(* Logix 5000 project; controller Lavado_Tapado Emulate 5570 rev 32.11; software revision 32.00 *)

TASK MainTask (continuous, watchdog 500 ms) : MainProgram

MODULES
   Local : Emulate 5570 (ICP 2, rev 32.11)
END_MODULES

VAR_GLOBAL   (* controller tags *)
   ACT_LLT_AlineadorLlenado : BOOL;   // Orden NX de extensión del alineador.
   ACT_LLT_Banda : BOOL := 1;   // Orden NX de encendido de la banda.
   ACT_LLT_BoquillaLlenado : BOOL;   // Orden NX de descenso de la boquilla.
   ACT_LLT_BorrarBotella : BOOL;   // Orden NX de borrar el CAD sin tapa.
   ACT_LLT_DetencionLlenado : BOOL;   // Orden NX de retención de botellas.
   ACT_LLT_NuevaBotella : BOOL;   // Orden NX de crear el CAD con tapa.
   ACT_LLT_PosicionamientoTapado : DINT;   // Consigna numérica NX del carrusel en grados.
   ACT_LLT_Remachadora : BOOL;   // Orden NX de descenso de la remachadora.
   CMD_LLT_Inicio : BOOL := 1;   // Botón momentáneo de Inicio desde Studio 5000.
   CMD_LLT_Parada : BOOL;   // Botón momentáneo de Parada; abandona el automático.
   CMD_LLT_Reinicio : BOOL;   // Botón momentáneo de Reinicio con prioridad máxima.
   CNT_LLT_BotellasGrupo : DINT; {access None}   // Conteo numérico del grupo de botellas.
   ET_LLT_000_Inicial : BOOL; {access None}   // Etapa 0 inicial y reiniciada.
   ET_LLT_010_Automatico : BOOL := 1; {access None}   // Etapa 10 de automático concurrente.
   ET_LLT_090_Parada : BOOL; {access None}   // Etapa 90 de parada sin reanudación.
   ET_LLT_100_Admision : BOOL := 1; {access None}   // Etapa 100 de admisión y conteo.
   ET_LLT_110_Posicionamiento : BOOL; {access None}   // Etapa 110 de posicionamiento durante 2 s.
   ET_LLT_120_Alineacion : BOOL; {access None}   // Etapa 120 de extensión del alineador.
   ET_LLT_130_DescensoBoquilla : BOOL; {access None}   // Etapa 130 de descenso de boquilla.
   ET_LLT_140_Llenado : BOOL; {access None}   // Etapa 140 de llenado durante 2 s.
   ET_LLT_150_RetiradaBoquilla : BOOL; {access None}   // Etapa 150 de subida de boquilla.
   ET_LLT_160_RetiradaAlineacion : BOOL; {access None}   // Etapa 160 de retracción del alineador.
   ET_LLT_170_Transferencia : BOOL; {access None}   // Etapa 170 de transferencia del grupo.
   ET_LLT_200_EsperaPrimeraBotella : BOOL; {access None}   // Etapa 200 de espera de primera botella en carrusel.
   ET_LLT_210_PrimerIndexado : BOOL; {access None}   // Etapa 210 de primer indexado.
   ET_LLT_220_BorrarPrimera : BOOL; {access None}   // Etapa 220 de borrar primera botella.
   ET_LLT_222_CrearPrimera : BOOL; {access None}   // Etapa 222 de crear primera botella con tapa.
   ET_LLT_230_SegundoIndexado : BOOL; {access None}   // Etapa 230 de segundo indexado.
   ET_LLT_240_Borrar : BOOL; {access None}   // Etapa 240 de borrado en rama paralela.
   ET_LLT_241_Crear : BOOL; {access None}   // Etapa 241 de creación en rama paralela.
   ET_LLT_242_TapadoListo : BOOL; {access None}   // Etapa 242 de tapado listo.
   ET_LLT_250_BajarRemachadora : BOOL; {access None}   // Etapa 250 de descenso de remachadora.
   ET_LLT_251_SubirRemachadora : BOOL; {access None}   // Etapa 251 de subida de remachadora.
   ET_LLT_252_RemachadoListo : BOOL; {access None}   // Etapa 252 de remachado listo.
   ET_LLT_260_IndexadoSincronizado : BOOL := 1; {access None}   // Etapa 260 de indexado sincronizado.
   FL_LLT_ContadorEntrada : BOOL; {access None}   // Pulso de flanco ascendente del sensor de entrada.
   FL_LLT_CuartaBotella : BOOL; {access None}   // Pulso de cuarto evento aceptado.
   IDX_LLT_Carrusel : DINT; {access None}   // Índice cíclico del carrusel de 0 a 4.
   M_LLT_ConteoHabilitado : BOOL := 1; {access None}   // Ventana de conteo exclusiva de etapa 100.
   M_LLT_ReinicioCumplido : BOOL := 1; {access None}   // Memoria que exige Reinicio después de Parada antes de aceptar Inicio.
   M_LLT_RemacheVioAusencia : BOOL := 1; {access None}   // Memoria de ausencia previa del sensor de remache.
   M_LLT_TapadoVioAusencia : BOOL := 1; {access None}   // Memoria de ausencia previa del sensor de tapado.
   MEM_LLT_ContadorEntradaPrev : BOOL; {access None}   // Memoria ONS global del sensor de entrada; evita contar un nivel ya activo al entrar en admisión.
   PAR_LLT_BotellasGrupo : DINT := 4;   // Cantidad objetivo de botellas por grupo.
   PAR_LLT_PasoCarrusel_deg : DINT := -72;   // Paso angular lógico del carrusel.
   PAR_LLT_PosicionesCarrusel : DINT := 5;   // Cantidad de posiciones lógicas del carrusel.
   PAR_LLT_T_Llenado_ms : DINT := 2000;   // Preset de llenado en milisegundos.
   PAR_LLT_T_Posicionamiento_ms : DINT := 2000;   // Preset de posicionamiento en milisegundos.
   SE_LLT_AgregarTapa : BOOL;   // Botella presente en la estación de tapado.
   SE_LLT_AlineacionLlenadoExtendido : BOOL;   // Alineador completamente extendido.
   SE_LLT_AlineacionLlenadoRetraido : BOOL := 1;   // Alineador completamente retraído.
   SE_LLT_BoquillaAbajo : BOOL;   // Boquilla completamente abajo.
   SE_LLT_BoquillaArriba : BOOL := 1;   // Boquilla completamente arriba.
   SE_LLT_ContadorEntrada : BOOL;   // Botella frente al sensor de entrada; se cuenta solo por flanco en admisión.
   SE_LLT_DeteccionBotellaTapado : BOOL;   // Botella disponible en la entrada del carrusel.
   SE_LLT_ParadaRemache : BOOL := 1;   // Botella presente en la estación de remache.
   SE_LLT_RemachadoraAbajo : BOOL;   // Remachadora completamente abajo.
   SE_LLT_RemachadoraArriba : BOOL := 1;   // Remachadora completamente arriba.
   SE_LLT_SinDetencion : BOOL := 1;   // Tope retirado y paso libre; no existe sensor de tope extendido.
   SP_LLT_Carrusel_deg : DINT; {access None}   // Consigna interna vigente del carrusel en grados.
   TM_LLT_Llenado : TIMER := (PRE := 2000); {access None}   // Temporizador de llenado de 2 s.
   TM_LLT_Posicionamiento : TIMER := (PRE := 2000); {access None}   // Temporizador de posicionamiento de 2 s.
   TR_LLT_t00 : BOOL; {access None}   // Snapshot de la transición t00; se evalúa antes de actualizar etapas.
   TR_LLT_t10 : BOOL; {access None}   // Snapshot de la transición t10; se evalúa antes de actualizar etapas.
   TR_LLT_t100 : BOOL; {access None}   // Snapshot de la transición t100; se evalúa antes de actualizar etapas.
   TR_LLT_t110 : BOOL; {access None}   // Snapshot de la transición t110; se evalúa antes de actualizar etapas.
   TR_LLT_t120 : BOOL; {access None}   // Snapshot de la transición t120; se evalúa antes de actualizar etapas.
   TR_LLT_t130 : BOOL; {access None}   // Snapshot de la transición t130; se evalúa antes de actualizar etapas.
   TR_LLT_t140 : BOOL; {access None}   // Snapshot de la transición t140; se evalúa antes de actualizar etapas.
   TR_LLT_t150 : BOOL; {access None}   // Snapshot de la transición t150; se evalúa antes de actualizar etapas.
   TR_LLT_t160 : BOOL; {access None}   // Snapshot de la transición t160; se evalúa antes de actualizar etapas.
   TR_LLT_t170 : BOOL; {access None}   // Snapshot de la transición t170; se evalúa antes de actualizar etapas.
   TR_LLT_t200 : BOOL; {access None}   // Snapshot de la transición t200; se evalúa antes de actualizar etapas.
   TR_LLT_t210 : BOOL; {access None}   // Snapshot de la transición t210; se evalúa antes de actualizar etapas.
   TR_LLT_t220 : BOOL; {access None}   // Snapshot de la transición t220; se evalúa antes de actualizar etapas.
   TR_LLT_t220a : BOOL; {access None}   // Snapshot de la transición t220a; se evalúa antes de actualizar etapas.
   TR_LLT_t230 : BOOL; {access None}   // Snapshot de la transición t230; se evalúa antes de actualizar etapas.
   TR_LLT_t240 : BOOL; {access None}   // Snapshot de la transición t240; se evalúa antes de actualizar etapas.
   TR_LLT_t240a : BOOL; {access None}   // Snapshot de la transición t240a; se evalúa antes de actualizar etapas.
   TR_LLT_t250 : BOOL; {access None}   // Snapshot de la transición t250; se evalúa antes de actualizar etapas.
   TR_LLT_t250a : BOOL; {access None}   // Snapshot de la transición t250a; se evalúa antes de actualizar etapas.
   TR_LLT_t260 : BOOL; {access None}   // Snapshot de la transición t260; se evalúa antes de actualizar etapas.
   TR_LLT_t261 : BOOL; {access None}   // Snapshot de la transición t261; se evalúa antes de actualizar etapas.
   TR_LLT_t90 : BOOL; {access None}   // Snapshot de la transición t90; se evalúa antes de actualizar etapas.
END_VAR

PROGRAM MainProgram   (* main routine MainRoutine *)

ROUTINE MainRoutine   (* ladder *)
// Despacha seis rutinas simplificadas en orden determinista.
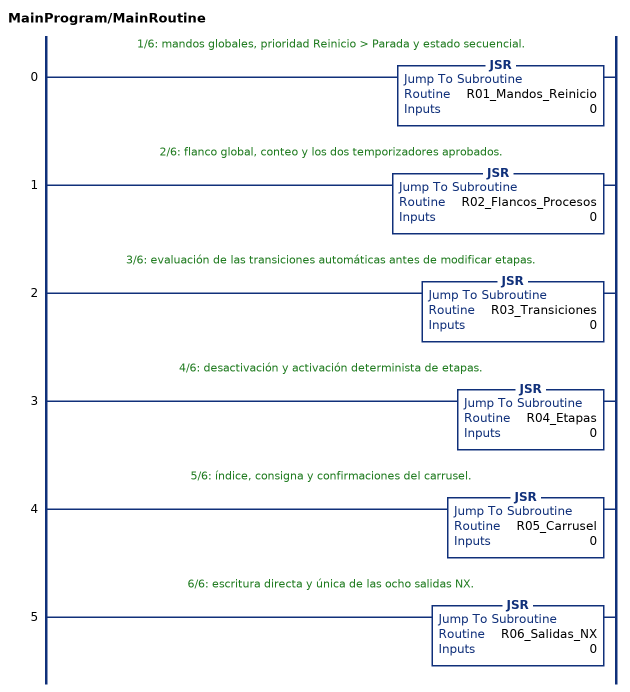
   // 1/6: mandos globales, prioridad Reinicio > Parada y estado secuencial.
   0: JSR(R01_Mandos_Reinicio,0);
   // 2/6: flanco global, conteo y los dos temporizadores aprobados.
   1: JSR(R02_Flancos_Procesos,0);
   // 3/6: evaluación de las transiciones automáticas antes de modificar etapas.
   2: JSR(R03_Transiciones,0);
   // 4/6: desactivación y activación determinista de etapas.
   3: JSR(R04_Etapas,0);
   // 5/6: índice, consigna y confirmaciones del carrusel.
   4: JSR(R05_Carrusel,0);
   // 6/6: escritura directa y única de las ocho salidas NX.
   5: JSR(R06_Salidas_NX,0);
END_ROUTINE

ROUTINE R01_Mandos_Reinicio   (* ladder *)
// Mandos globales y retorno simple al estado inicial sin escribir actuadores.
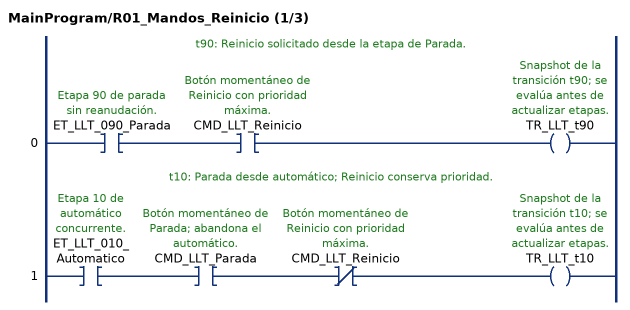
   // t90: Reinicio solicitado desde la etapa de Parada.
   0: XIC(ET_LLT_090_Parada)XIC(CMD_LLT_Reinicio)OTE(TR_LLT_t90);
   // t10: Parada desde automático; Reinicio conserva prioridad.
   1: XIC(ET_LLT_010_Automatico)XIC(CMD_LLT_Parada)XIO(CMD_LLT_Reinicio)OTE(TR_LLT_t10);
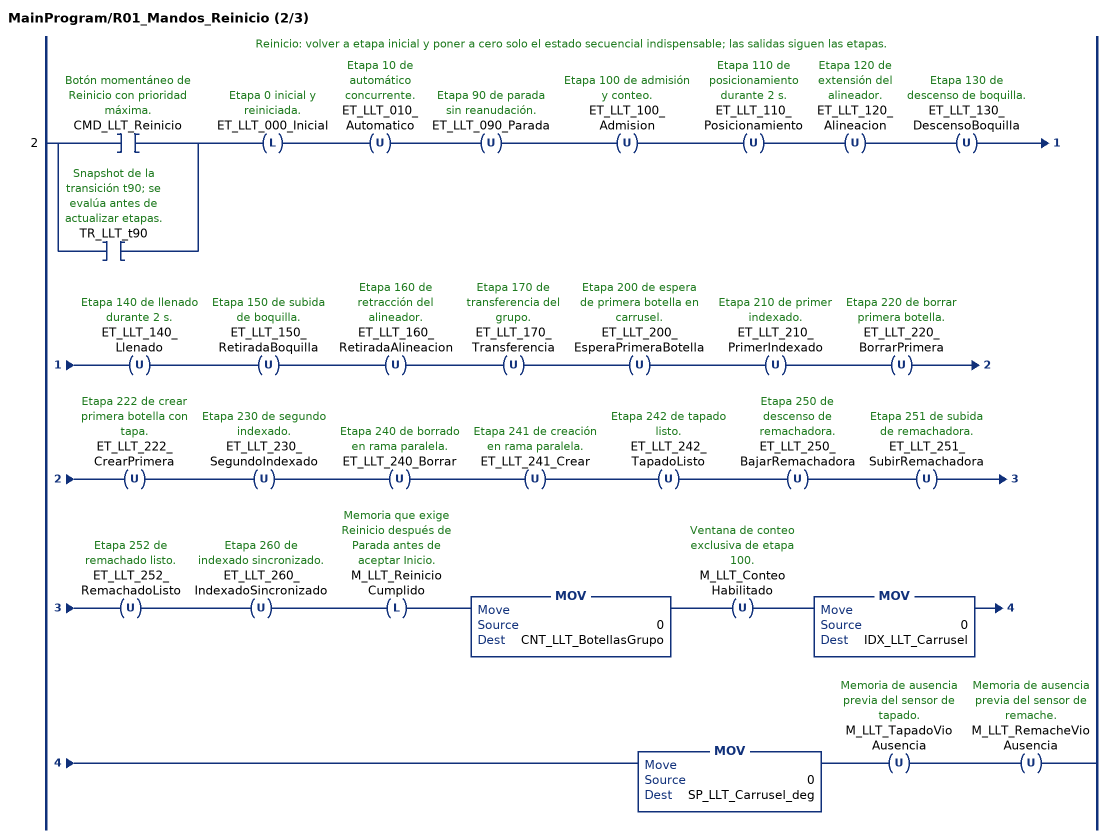
   // Reinicio: volver a etapa inicial y poner a cero solo el estado secuencial indispensable; las salidas siguen las etapas.
   2: [XIC(CMD_LLT_Reinicio) ,XIC(TR_LLT_t90) ]OTL(ET_LLT_000_Inicial)OTU(ET_LLT_010_Automatico)OTU(ET_LLT_090_Parada)OTU(ET_LLT_100_Admision)OTU(ET_LLT_110_Posicionamiento)OTU(ET_LLT_120_Alineacion)OTU(ET_LLT_130_DescensoBoquilla)OTU(ET_LLT_140_Llenado)OTU(ET_LLT_150_RetiradaBoquilla)OTU(ET_LLT_160_RetiradaAlineacion)OTU(ET_LLT_170_Transferencia)OTU(ET_LLT_200_EsperaPrimeraBotella)OTU(ET_LLT_210_PrimerIndexado)OTU(ET_LLT_220_BorrarPrimera)OTU(ET_LLT_222_CrearPrimera)OTU(ET_LLT_230_SegundoIndexado)OTU(ET_LLT_240_Borrar)OTU(ET_LLT_241_Crear)OTU(ET_LLT_242_TapadoListo)OTU(ET_LLT_250_BajarRemachadora)OTU(ET_LLT_251_SubirRemachadora)OTU(ET_LLT_252_RemachadoListo)OTU(ET_LLT_260_IndexadoSincronizado)OTL(M_LLT_ReinicioCumplido)MOV(0,CNT_LLT_BotellasGrupo)OTU(M_LLT_ConteoHabilitado)MOV(0,IDX_LLT_Carrusel)MOV(0,SP_LLT_Carrusel_deg)OTU(M_LLT_TapadoVioAusencia)OTU(M_LLT_RemacheVioAusencia);
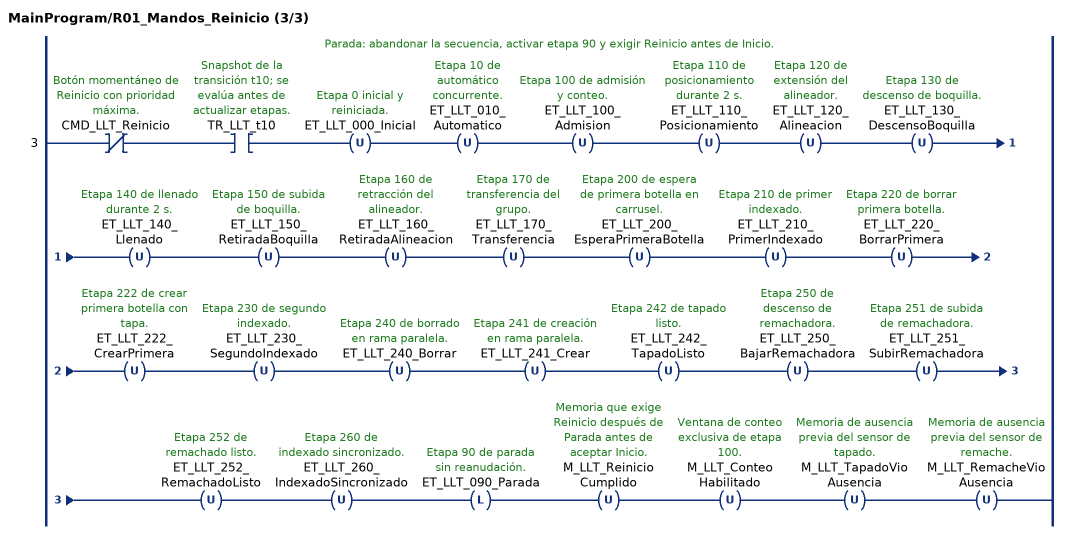
   // Parada: abandonar la secuencia, activar etapa 90 y exigir Reinicio antes de Inicio.
   3: XIO(CMD_LLT_Reinicio)XIC(TR_LLT_t10)OTU(ET_LLT_000_Inicial)OTU(ET_LLT_010_Automatico)OTU(ET_LLT_100_Admision)OTU(ET_LLT_110_Posicionamiento)OTU(ET_LLT_120_Alineacion)OTU(ET_LLT_130_DescensoBoquilla)OTU(ET_LLT_140_Llenado)OTU(ET_LLT_150_RetiradaBoquilla)OTU(ET_LLT_160_RetiradaAlineacion)OTU(ET_LLT_170_Transferencia)OTU(ET_LLT_200_EsperaPrimeraBotella)OTU(ET_LLT_210_PrimerIndexado)OTU(ET_LLT_220_BorrarPrimera)OTU(ET_LLT_222_CrearPrimera)OTU(ET_LLT_230_SegundoIndexado)OTU(ET_LLT_240_Borrar)OTU(ET_LLT_241_Crear)OTU(ET_LLT_242_TapadoListo)OTU(ET_LLT_250_BajarRemachadora)OTU(ET_LLT_251_SubirRemachadora)OTU(ET_LLT_252_RemachadoListo)OTU(ET_LLT_260_IndexadoSincronizado)OTL(ET_LLT_090_Parada)OTU(M_LLT_ReinicioCumplido)OTU(M_LLT_ConteoHabilitado)OTU(M_LLT_TapadoVioAusencia)OTU(M_LLT_RemacheVioAusencia);
END_ROUTINE

ROUTINE R02_Flancos_Procesos   (* ladder *)
// Flanco global, conteo de cuatro y únicamente dos TON.
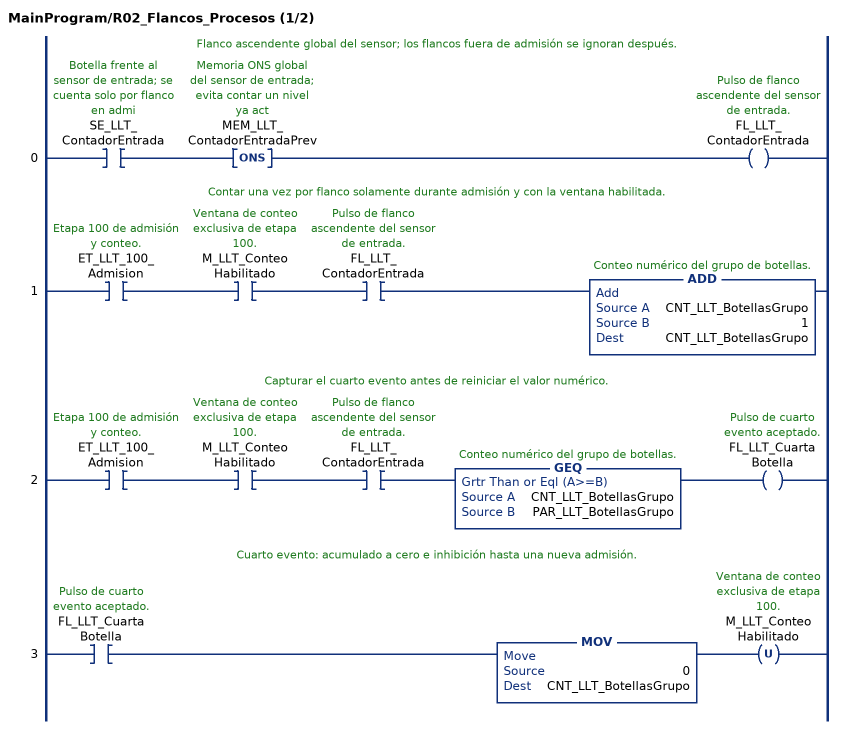
   // Flanco ascendente global del sensor; los flancos fuera de admisión se ignoran después.
   0: XIC(SE_LLT_ContadorEntrada)ONS(MEM_LLT_ContadorEntradaPrev)OTE(FL_LLT_ContadorEntrada);
   // Contar una vez por flanco solamente durante admisión y con la ventana habilitada.
   1: XIC(ET_LLT_100_Admision)XIC(M_LLT_ConteoHabilitado)XIC(FL_LLT_ContadorEntrada)ADD(CNT_LLT_BotellasGrupo,1,CNT_LLT_BotellasGrupo);
   // Capturar el cuarto evento antes de reiniciar el valor numérico.
   2: XIC(ET_LLT_100_Admision)XIC(M_LLT_ConteoHabilitado)XIC(FL_LLT_ContadorEntrada)GEQ(CNT_LLT_BotellasGrupo,PAR_LLT_BotellasGrupo)OTE(FL_LLT_CuartaBotella);
   // Cuarto evento: acumulado a cero e inhibición hasta una nueva admisión.
   3: XIC(FL_LLT_CuartaBotella)MOV(0,CNT_LLT_BotellasGrupo)OTU(M_LLT_ConteoHabilitado);
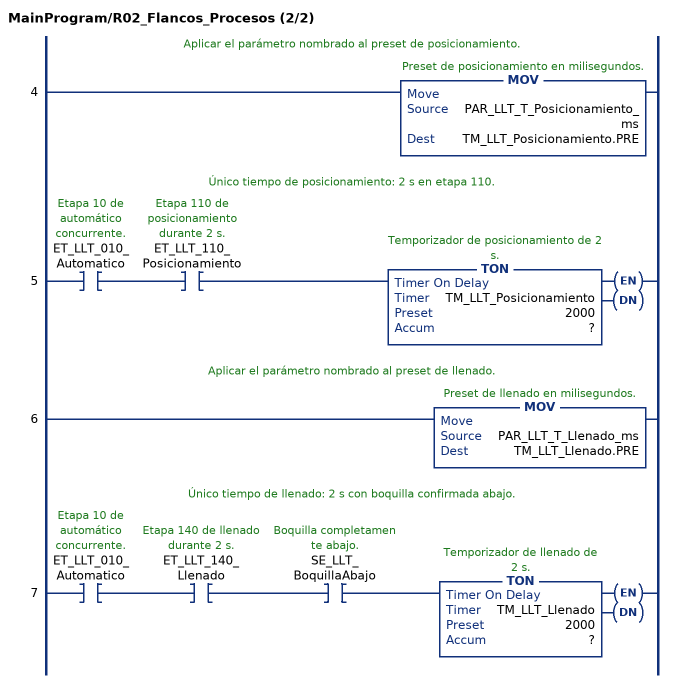
   // Aplicar el parámetro nombrado al preset de posicionamiento.
   4: MOV(PAR_LLT_T_Posicionamiento_ms,TM_LLT_Posicionamiento.PRE);
   // Único tiempo de posicionamiento: 2 s en etapa 110.
   5: XIC(ET_LLT_010_Automatico)XIC(ET_LLT_110_Posicionamiento)TON(TM_LLT_Posicionamiento,?,?);
   // Aplicar el parámetro nombrado al preset de llenado.
   6: MOV(PAR_LLT_T_Llenado_ms,TM_LLT_Llenado.PRE);
   // Único tiempo de llenado: 2 s con boquilla confirmada abajo.
   7: XIC(ET_LLT_010_Automatico)XIC(ET_LLT_140_Llenado)XIC(SE_LLT_BoquillaAbajo)TON(TM_LLT_Llenado,?,?);
END_ROUTINE

ROUTINE R03_Transiciones   (* ladder *)
// Evalúa las veinte transiciones automáticas; t10 y t90 se resuelven antes en mandos.
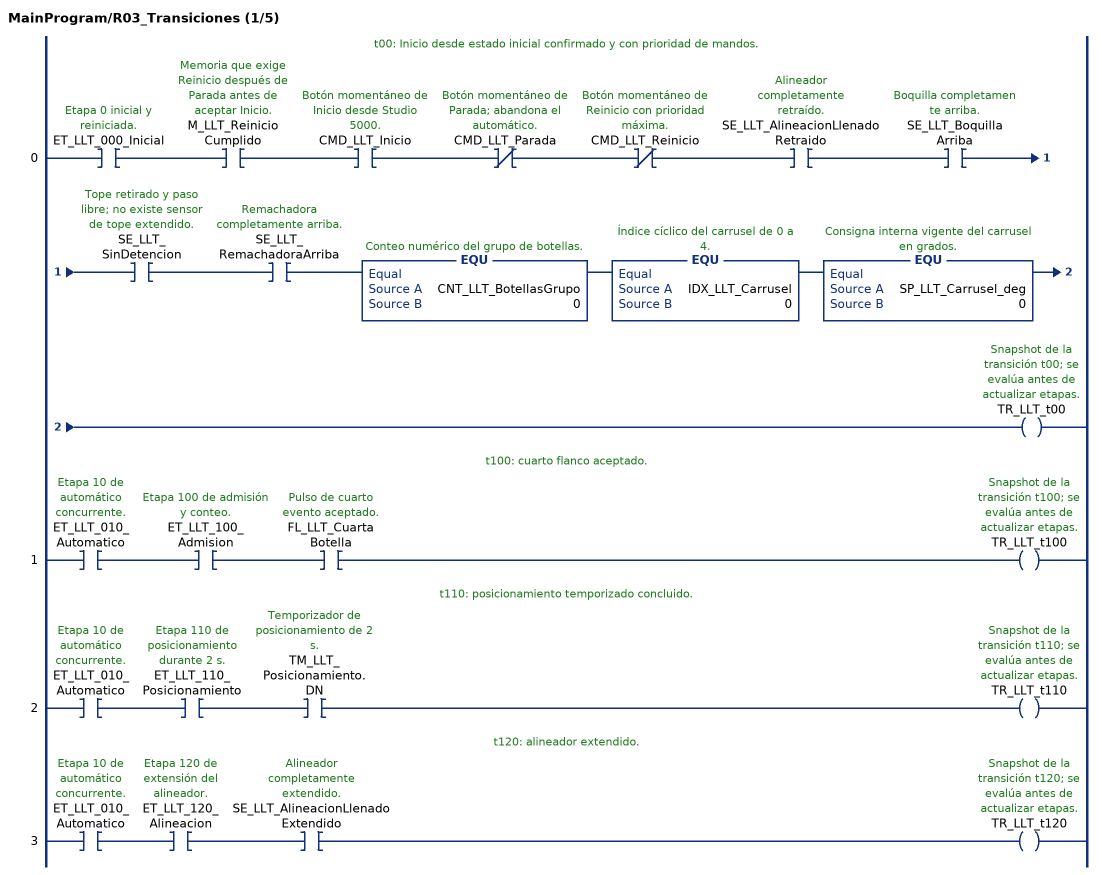
   // t00: Inicio desde estado inicial confirmado y con prioridad de mandos.
   0: XIC(ET_LLT_000_Inicial)XIC(M_LLT_ReinicioCumplido)XIC(CMD_LLT_Inicio)XIO(CMD_LLT_Parada)XIO(CMD_LLT_Reinicio)XIC(SE_LLT_AlineacionLlenadoRetraido)XIC(SE_LLT_BoquillaArriba)XIC(SE_LLT_SinDetencion)XIC(SE_LLT_RemachadoraArriba)EQU(CNT_LLT_BotellasGrupo,0)EQU(IDX_LLT_Carrusel,0)EQU(SP_LLT_Carrusel_deg,0)OTE(TR_LLT_t00);
   // t100: cuarto flanco aceptado.
   1: XIC(ET_LLT_010_Automatico)XIC(ET_LLT_100_Admision)XIC(FL_LLT_CuartaBotella)OTE(TR_LLT_t100);
   // t110: posicionamiento temporizado concluido.
   2: XIC(ET_LLT_010_Automatico)XIC(ET_LLT_110_Posicionamiento)XIC(TM_LLT_Posicionamiento.DN)OTE(TR_LLT_t110);
   // t120: alineador extendido.
   3: XIC(ET_LLT_010_Automatico)XIC(ET_LLT_120_Alineacion)XIC(SE_LLT_AlineacionLlenadoExtendido)OTE(TR_LLT_t120);
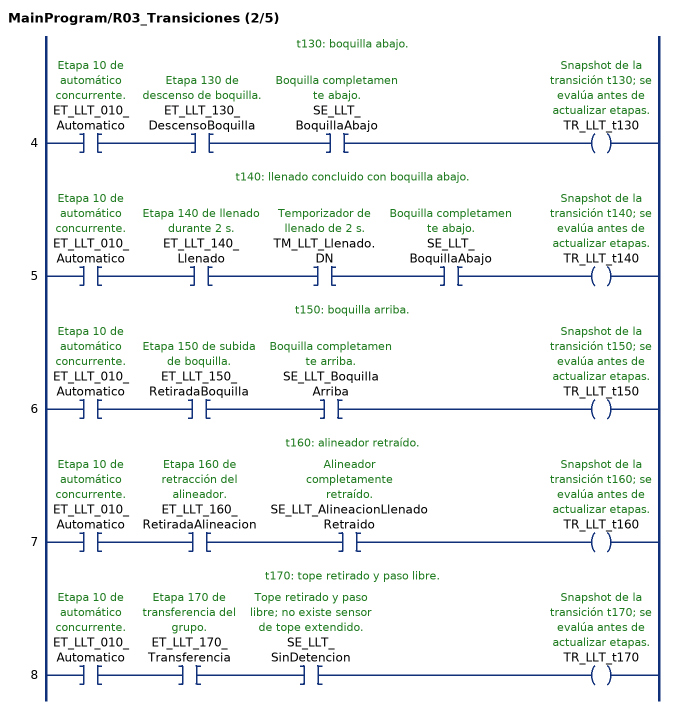
   // t130: boquilla abajo.
   4: XIC(ET_LLT_010_Automatico)XIC(ET_LLT_130_DescensoBoquilla)XIC(SE_LLT_BoquillaAbajo)OTE(TR_LLT_t130);
   // t140: llenado concluido con boquilla abajo.
   5: XIC(ET_LLT_010_Automatico)XIC(ET_LLT_140_Llenado)XIC(TM_LLT_Llenado.DN)XIC(SE_LLT_BoquillaAbajo)OTE(TR_LLT_t140);
   // t150: boquilla arriba.
   6: XIC(ET_LLT_010_Automatico)XIC(ET_LLT_150_RetiradaBoquilla)XIC(SE_LLT_BoquillaArriba)OTE(TR_LLT_t150);
   // t160: alineador retraído.
   7: XIC(ET_LLT_010_Automatico)XIC(ET_LLT_160_RetiradaAlineacion)XIC(SE_LLT_AlineacionLlenadoRetraido)OTE(TR_LLT_t160);
   // t170: tope retirado y paso libre.
   8: XIC(ET_LLT_010_Automatico)XIC(ET_LLT_170_Transferencia)XIC(SE_LLT_SinDetencion)OTE(TR_LLT_t170);
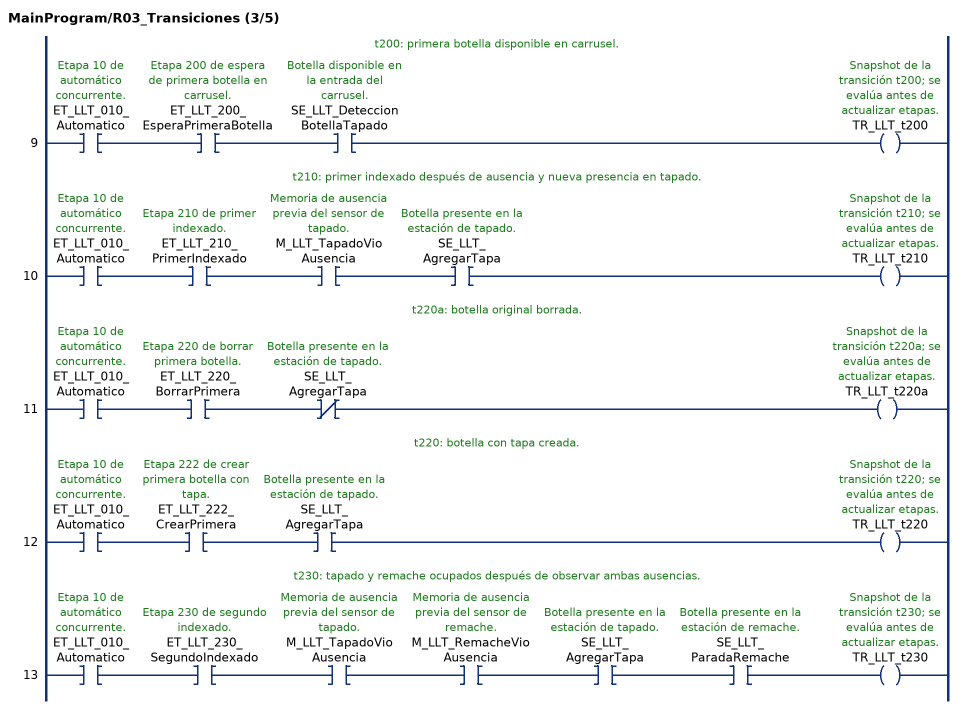
   // t200: primera botella disponible en carrusel.
   9: XIC(ET_LLT_010_Automatico)XIC(ET_LLT_200_EsperaPrimeraBotella)XIC(SE_LLT_DeteccionBotellaTapado)OTE(TR_LLT_t200);
   // t210: primer indexado después de ausencia y nueva presencia en tapado.
   10: XIC(ET_LLT_010_Automatico)XIC(ET_LLT_210_PrimerIndexado)XIC(M_LLT_TapadoVioAusencia)XIC(SE_LLT_AgregarTapa)OTE(TR_LLT_t210);
   // t220a: botella original borrada.
   11: XIC(ET_LLT_010_Automatico)XIC(ET_LLT_220_BorrarPrimera)XIO(SE_LLT_AgregarTapa)OTE(TR_LLT_t220a);
   // t220: botella con tapa creada.
   12: XIC(ET_LLT_010_Automatico)XIC(ET_LLT_222_CrearPrimera)XIC(SE_LLT_AgregarTapa)OTE(TR_LLT_t220);
   // t230: tapado y remache ocupados después de observar ambas ausencias.
   13: XIC(ET_LLT_010_Automatico)XIC(ET_LLT_230_SegundoIndexado)XIC(M_LLT_TapadoVioAusencia)XIC(M_LLT_RemacheVioAusencia)XIC(SE_LLT_AgregarTapa)XIC(SE_LLT_ParadaRemache)OTE(TR_LLT_t230);
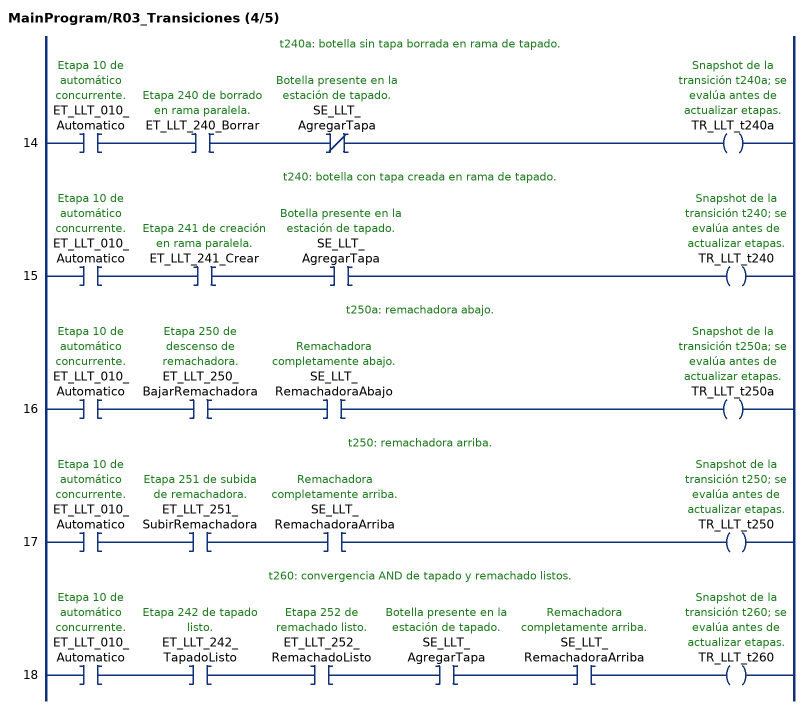
   // t240a: botella sin tapa borrada en rama de tapado.
   14: XIC(ET_LLT_010_Automatico)XIC(ET_LLT_240_Borrar)XIO(SE_LLT_AgregarTapa)OTE(TR_LLT_t240a);
   // t240: botella con tapa creada en rama de tapado.
   15: XIC(ET_LLT_010_Automatico)XIC(ET_LLT_241_Crear)XIC(SE_LLT_AgregarTapa)OTE(TR_LLT_t240);
   // t250a: remachadora abajo.
   16: XIC(ET_LLT_010_Automatico)XIC(ET_LLT_250_BajarRemachadora)XIC(SE_LLT_RemachadoraAbajo)OTE(TR_LLT_t250a);
   // t250: remachadora arriba.
   17: XIC(ET_LLT_010_Automatico)XIC(ET_LLT_251_SubirRemachadora)XIC(SE_LLT_RemachadoraArriba)OTE(TR_LLT_t250);
   // t260: convergencia AND de tapado y remachado listos.
   18: XIC(ET_LLT_010_Automatico)XIC(ET_LLT_242_TapadoListo)XIC(ET_LLT_252_RemachadoListo)XIC(SE_LLT_AgregarTapa)XIC(SE_LLT_RemachadoraArriba)OTE(TR_LLT_t260);
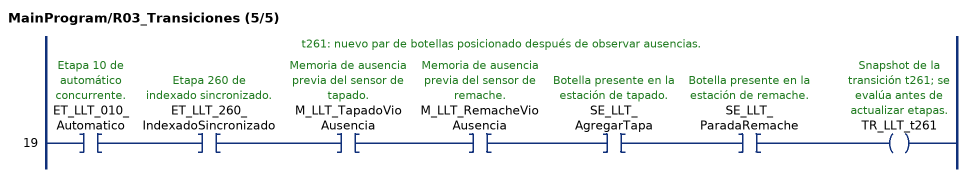
   // t261: nuevo par de botellas posicionado después de observar ausencias.
   19: XIC(ET_LLT_010_Automatico)XIC(ET_LLT_260_IndexadoSincronizado)XIC(M_LLT_TapadoVioAusencia)XIC(M_LLT_RemacheVioAusencia)XIC(SE_LLT_AgregarTapa)XIC(SE_LLT_ParadaRemache)OTE(TR_LLT_t261);
END_ROUTINE

ROUTINE R04_Etapas   (* ladder *)
// Actualiza etapas solamente después de evaluar todas las transiciones.
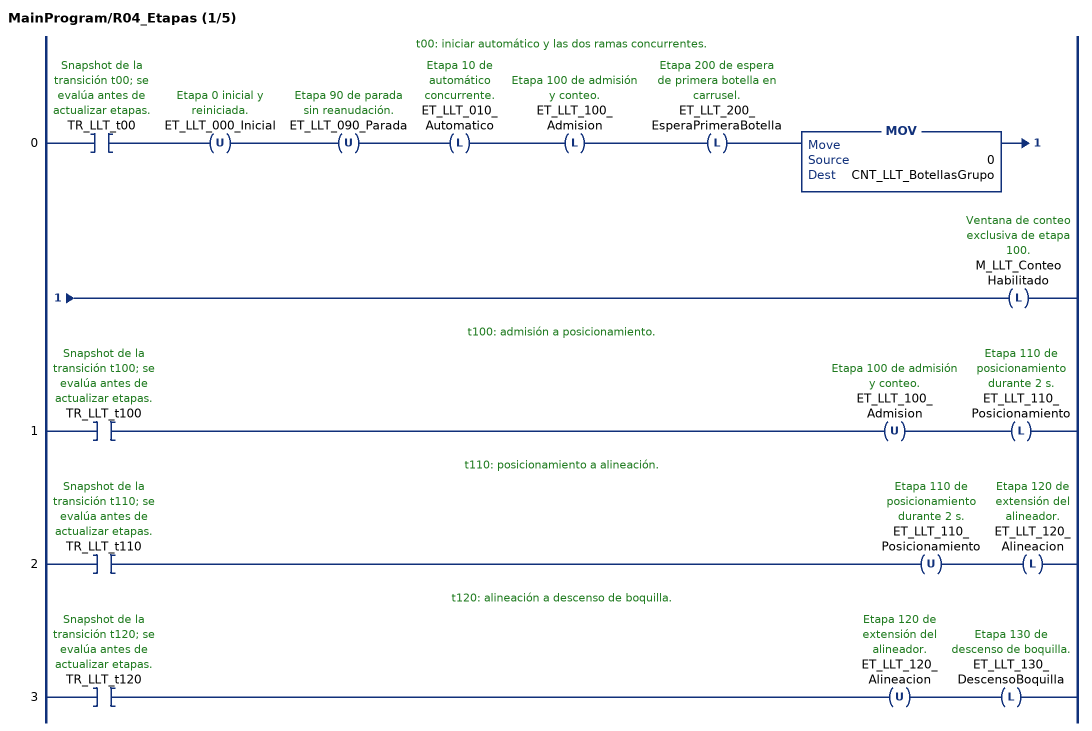
   // t00: iniciar automático y las dos ramas concurrentes.
   0: XIC(TR_LLT_t00)OTU(ET_LLT_000_Inicial)OTU(ET_LLT_090_Parada)OTL(ET_LLT_010_Automatico)OTL(ET_LLT_100_Admision)OTL(ET_LLT_200_EsperaPrimeraBotella)MOV(0,CNT_LLT_BotellasGrupo)OTL(M_LLT_ConteoHabilitado);
   // t100: admisión a posicionamiento.
   1: XIC(TR_LLT_t100)OTU(ET_LLT_100_Admision)OTL(ET_LLT_110_Posicionamiento);
   // t110: posicionamiento a alineación.
   2: XIC(TR_LLT_t110)OTU(ET_LLT_110_Posicionamiento)OTL(ET_LLT_120_Alineacion);
   // t120: alineación a descenso de boquilla.
   3: XIC(TR_LLT_t120)OTU(ET_LLT_120_Alineacion)OTL(ET_LLT_130_DescensoBoquilla);
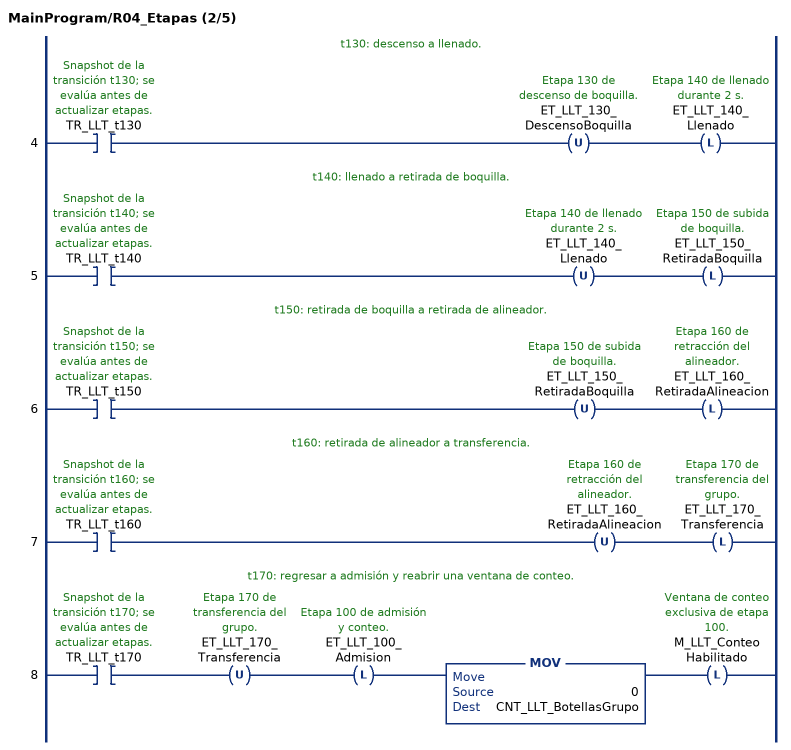
   // t130: descenso a llenado.
   4: XIC(TR_LLT_t130)OTU(ET_LLT_130_DescensoBoquilla)OTL(ET_LLT_140_Llenado);
   // t140: llenado a retirada de boquilla.
   5: XIC(TR_LLT_t140)OTU(ET_LLT_140_Llenado)OTL(ET_LLT_150_RetiradaBoquilla);
   // t150: retirada de boquilla a retirada de alineador.
   6: XIC(TR_LLT_t150)OTU(ET_LLT_150_RetiradaBoquilla)OTL(ET_LLT_160_RetiradaAlineacion);
   // t160: retirada de alineador a transferencia.
   7: XIC(TR_LLT_t160)OTU(ET_LLT_160_RetiradaAlineacion)OTL(ET_LLT_170_Transferencia);
   // t170: regresar a admisión y reabrir una ventana de conteo.
   8: XIC(TR_LLT_t170)OTU(ET_LLT_170_Transferencia)OTL(ET_LLT_100_Admision)MOV(0,CNT_LLT_BotellasGrupo)OTL(M_LLT_ConteoHabilitado);
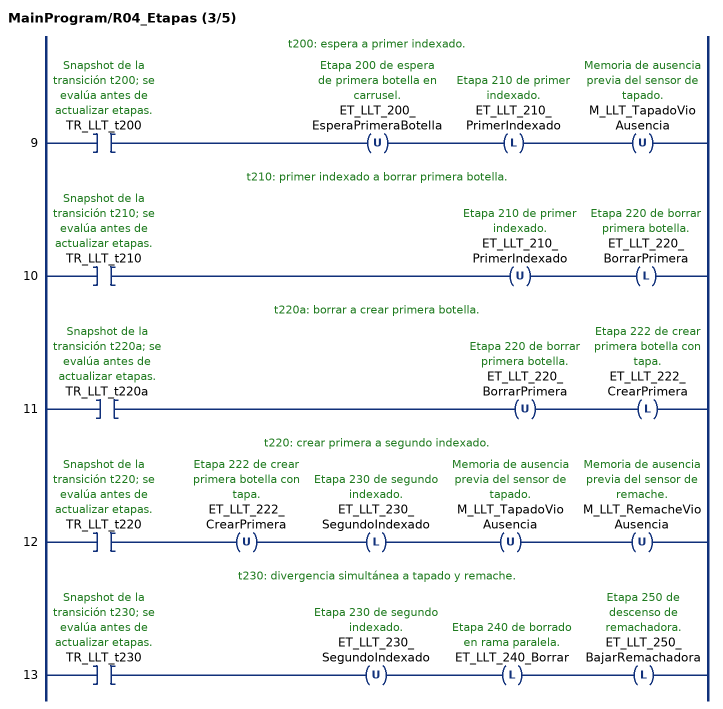
   // t200: espera a primer indexado.
   9: XIC(TR_LLT_t200)OTU(ET_LLT_200_EsperaPrimeraBotella)OTL(ET_LLT_210_PrimerIndexado)OTU(M_LLT_TapadoVioAusencia);
   // t210: primer indexado a borrar primera botella.
   10: XIC(TR_LLT_t210)OTU(ET_LLT_210_PrimerIndexado)OTL(ET_LLT_220_BorrarPrimera);
   // t220a: borrar a crear primera botella.
   11: XIC(TR_LLT_t220a)OTU(ET_LLT_220_BorrarPrimera)OTL(ET_LLT_222_CrearPrimera);
   // t220: crear primera a segundo indexado.
   12: XIC(TR_LLT_t220)OTU(ET_LLT_222_CrearPrimera)OTL(ET_LLT_230_SegundoIndexado)OTU(M_LLT_TapadoVioAusencia)OTU(M_LLT_RemacheVioAusencia);
   // t230: divergencia simultánea a tapado y remache.
   13: XIC(TR_LLT_t230)OTU(ET_LLT_230_SegundoIndexado)OTL(ET_LLT_240_Borrar)OTL(ET_LLT_250_BajarRemachadora);
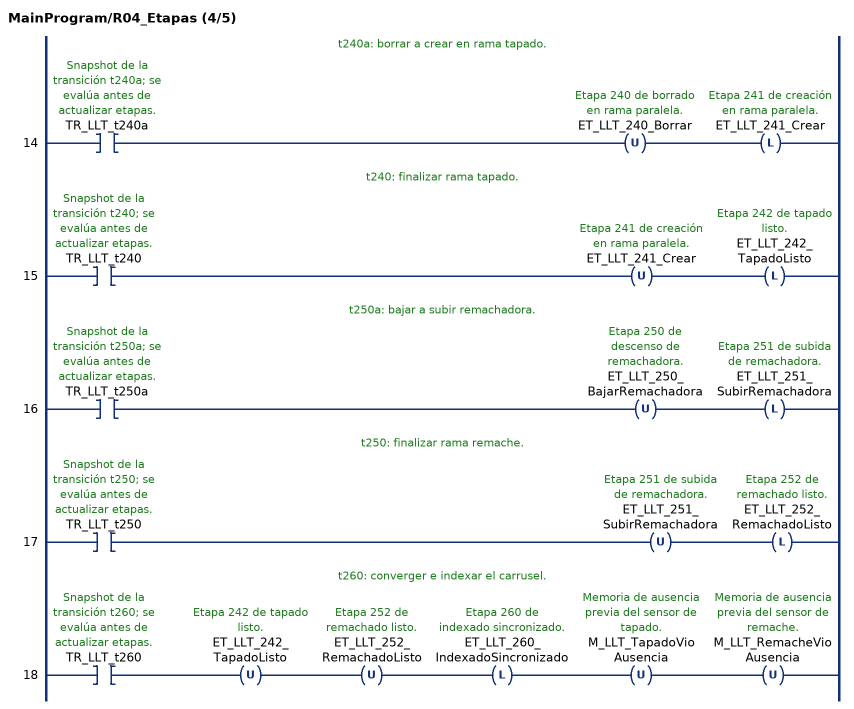
   // t240a: borrar a crear en rama tapado.
   14: XIC(TR_LLT_t240a)OTU(ET_LLT_240_Borrar)OTL(ET_LLT_241_Crear);
   // t240: finalizar rama tapado.
   15: XIC(TR_LLT_t240)OTU(ET_LLT_241_Crear)OTL(ET_LLT_242_TapadoListo);
   // t250a: bajar a subir remachadora.
   16: XIC(TR_LLT_t250a)OTU(ET_LLT_250_BajarRemachadora)OTL(ET_LLT_251_SubirRemachadora);
   // t250: finalizar rama remache.
   17: XIC(TR_LLT_t250)OTU(ET_LLT_251_SubirRemachadora)OTL(ET_LLT_252_RemachadoListo);
   // t260: converger e indexar el carrusel.
   18: XIC(TR_LLT_t260)OTU(ET_LLT_242_TapadoListo)OTU(ET_LLT_252_RemachadoListo)OTL(ET_LLT_260_IndexadoSincronizado)OTU(M_LLT_TapadoVioAusencia)OTU(M_LLT_RemacheVioAusencia);
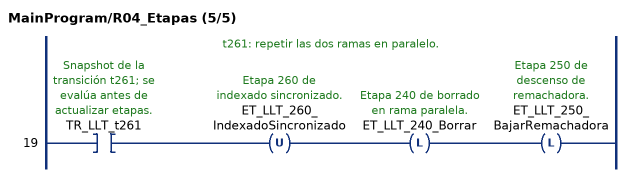
   // t261: repetir las dos ramas en paralelo.
   19: XIC(TR_LLT_t261)OTU(ET_LLT_260_IndexadoSincronizado)OTL(ET_LLT_240_Borrar)OTL(ET_LLT_250_BajarRemachadora);
END_ROUTINE

ROUTINE R05_Carrusel   (* ladder *)
// Actualización directa por pulso de transición, sin bit EV intermedio.
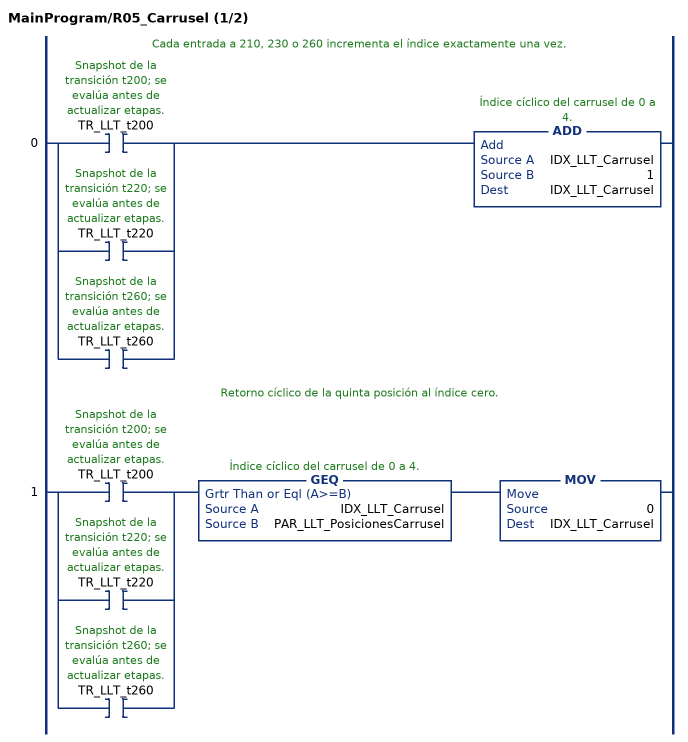
   // Cada entrada a 210, 230 o 260 incrementa el índice exactamente una vez.
   0: [XIC(TR_LLT_t200) ,XIC(TR_LLT_t220) ,XIC(TR_LLT_t260) ]ADD(IDX_LLT_Carrusel,1,IDX_LLT_Carrusel);
   // Retorno cíclico de la quinta posición al índice cero.
   1: [XIC(TR_LLT_t200) ,XIC(TR_LLT_t220) ,XIC(TR_LLT_t260) ]GEQ(IDX_LLT_Carrusel,PAR_LLT_PosicionesCarrusel)MOV(0,IDX_LLT_Carrusel);
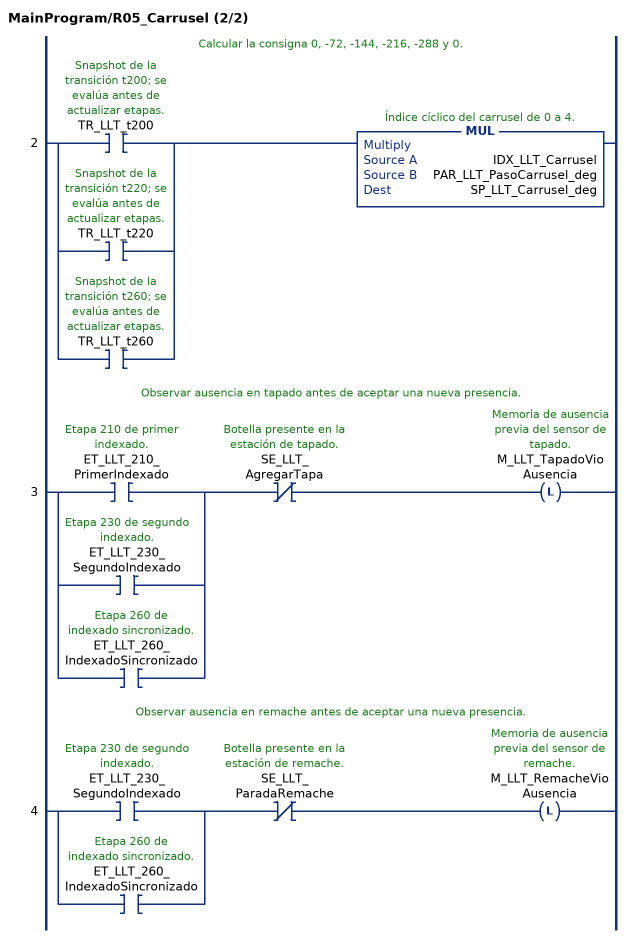
   // Calcular la consigna 0, -72, -144, -216, -288 y 0.
   2: [XIC(TR_LLT_t200) ,XIC(TR_LLT_t220) ,XIC(TR_LLT_t260) ]MUL(IDX_LLT_Carrusel,PAR_LLT_PasoCarrusel_deg,SP_LLT_Carrusel_deg);
   // Observar ausencia en tapado antes de aceptar una nueva presencia.
   3: [XIC(ET_LLT_210_PrimerIndexado) ,XIC(ET_LLT_230_SegundoIndexado) ,XIC(ET_LLT_260_IndexadoSincronizado) ]XIO(SE_LLT_AgregarTapa)OTL(M_LLT_TapadoVioAusencia);
   // Observar ausencia en remache antes de aceptar una nueva presencia.
   4: [XIC(ET_LLT_230_SegundoIndexado) ,XIC(ET_LLT_260_IndexadoSincronizado) ]XIO(SE_LLT_ParadaRemache)OTL(M_LLT_RemacheVioAusencia);
END_ROUTINE

ROUTINE R06_Salidas_NX   (* ladder *)
// Las etapas escriben directamente una sola vez cada salida NX.
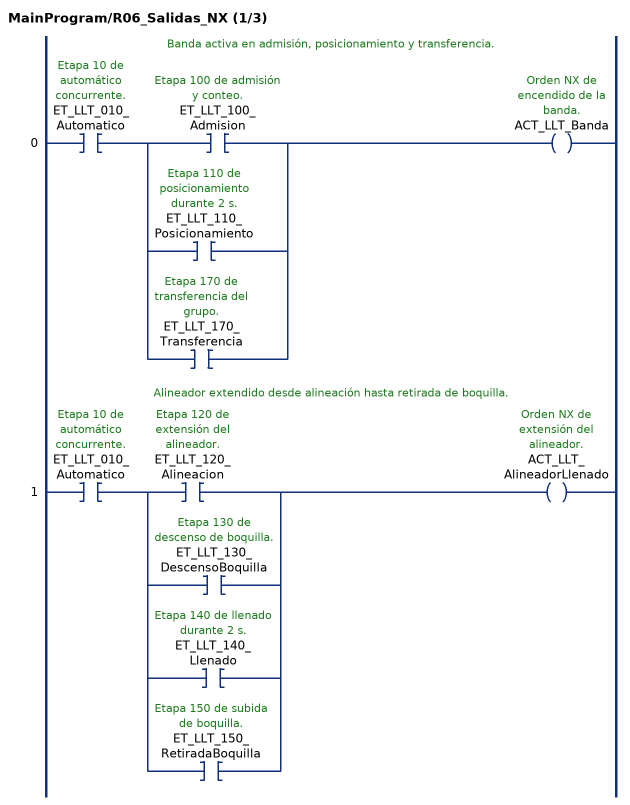
   // Banda activa en admisión, posicionamiento y transferencia.
   0: XIC(ET_LLT_010_Automatico)[XIC(ET_LLT_100_Admision) ,XIC(ET_LLT_110_Posicionamiento) ,XIC(ET_LLT_170_Transferencia) ]OTE(ACT_LLT_Banda);
   // Alineador extendido desde alineación hasta retirada de boquilla.
   1: XIC(ET_LLT_010_Automatico)[XIC(ET_LLT_120_Alineacion) ,XIC(ET_LLT_130_DescensoBoquilla) ,XIC(ET_LLT_140_Llenado) ,XIC(ET_LLT_150_RetiradaBoquilla) ]OTE(ACT_LLT_AlineadorLlenado);
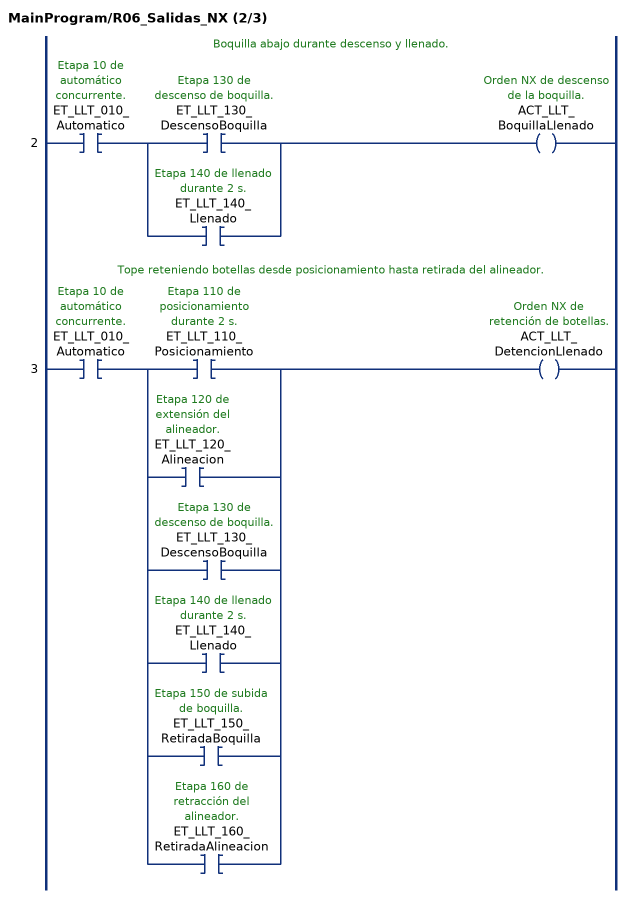
   // Boquilla abajo durante descenso y llenado.
   2: XIC(ET_LLT_010_Automatico)[XIC(ET_LLT_130_DescensoBoquilla) ,XIC(ET_LLT_140_Llenado) ]OTE(ACT_LLT_BoquillaLlenado);
   // Tope reteniendo botellas desde posicionamiento hasta retirada del alineador.
   3: XIC(ET_LLT_010_Automatico)[XIC(ET_LLT_110_Posicionamiento) ,XIC(ET_LLT_120_Alineacion) ,XIC(ET_LLT_130_DescensoBoquilla) ,XIC(ET_LLT_140_Llenado) ,XIC(ET_LLT_150_RetiradaBoquilla) ,XIC(ET_LLT_160_RetiradaAlineacion) ]OTE(ACT_LLT_DetencionLlenado);
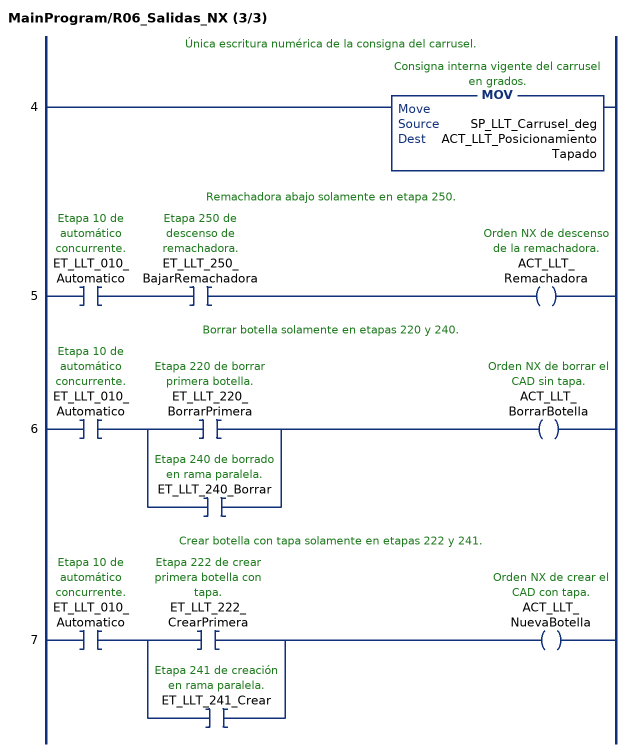
   // Única escritura numérica de la consigna del carrusel.
   4: MOV(SP_LLT_Carrusel_deg,ACT_LLT_PosicionamientoTapado);
   // Remachadora abajo solamente en etapa 250.
   5: XIC(ET_LLT_010_Automatico)XIC(ET_LLT_250_BajarRemachadora)OTE(ACT_LLT_Remachadora);
   // Borrar botella solamente en etapas 220 y 240.
   6: XIC(ET_LLT_010_Automatico)[XIC(ET_LLT_220_BorrarPrimera) ,XIC(ET_LLT_240_Borrar) ]OTE(ACT_LLT_BorrarBotella);
   // Crear botella con tapa solamente en etapas 222 y 241.
   7: XIC(ET_LLT_010_Automatico)[XIC(ET_LLT_222_CrearPrimera) ,XIC(ET_LLT_241_Crear) ]OTE(ACT_LLT_NuevaBotella);
END_ROUTINE
END_PROGRAM
